KUKA KRL program: makrosps6.src

&ACCESS RV
&PARAM TEMPLATE = C:\KRC\Roboter\Template\makrospsvorgabe.src
&PARAM EDITMASK = MakroSPS6
&PARAM TPVW_VERSION=8.3.17
DEF MAKROSPS6 ( )
; FOLD Makro Anfang;%{PSE} %MKUKATPVW
SPS_N=-1
; ENDFOLD
; FOLD ;%{H}
END
; ENDFOLD
